// TwinCAT 3 PLC project TcoDataTests
// Title: TcoDataTests
// Company: Vortex.Library
// ProjectVersion: 0.6.0.913
// ProgramVersion: 3.1.4024.12
// libraries:
//   Tc2_Standard, * (Beckhoff Automation GmbH)
//   Tc2_System, * (Beckhoff Automation GmbH)
//   Tc3_Module, * (Beckhoff Automation GmbH)
//   TcoCore, 0.6.0.913 (Vortex.Library)
//   TcoData, 0.6.0.913 (Vortex.Library)
// project tree:
//   DUTs/ SampleDataStructureLevel2.TcDUT, SampleDataStructure.TcDUT
//   / PlcTask.TcTTO
//   POUs/Data/ DataManager.TcPOU, eDataTests.TcDUT, TcoDataExchangeTests.TcPOU
//   POUs/Data/_dummyData/ enumStations.TcDUT, fbAnalogueValueData.TcDUT, stAnalogueProcessData.TcDUT, stCu_Header.TcDUT, stCu_ProcessData.TcDUT, stCu_ProcessDataBase.TcDUT, stEntityHeader.TcDUT, stProcessData.TcDUT
//   POUs/Examples/ eExamplesStates.TcDUT, SandboxData_Plc1.TcDUT, stProcessData_Plc1.TcDUT, stProcessData_Plc2.TcDUT, TcoDataManagerPlc1.TcPOU, TcoDataManagerPlc2.TcPOU, SandboxData.TcDUT, SandboxContext.TcPOU, TcoDataManager.TcPOU
//   POUs/ MAIN.TcPOU, TestDataContext.TcPOU
// (motion and I/O tree: see PLC project tcodata)
// real-time tasks:
//   TASK PlcTask: cycle T#10ms, priority 20, ADS port 350

CONFIGURATION TcoDataTests
    RESOURCE PLC ON TwinCAT3
        TASK PlcTask(INTERVAL := T#10ms, PRIORITY := 20);
        PROGRAM MAIN WITH PlcTask : MAIN;
    END_RESOURCE
END_CONFIGURATION

// ---- DUTs/SampleDataStructureLevel2.TcDUT
TYPE SampleDataStructureLevel2 :
STRUCT
    SampleString : STRING;
    SampleString2 : STRING := '32432423tewtew*-+/';
    SampleInt : INT;
    SampleBool : BOOL;
    SampleBool2 : BOOL := TRUE;
    SampleWString : WSTRING;
    SampleLREAL : LREAL;
END_STRUCT
END_TYPE

// ---- DUTs/SampleDataStructure.TcDUT
TYPE SampleDataStructure :
STRUCT
    SampleString : STRING;
    SampleString2 : STRING := '3retewtertert2342345*-+/';
    SampleInt : INT;
    SampleInt2 : INT := 432;
    SampleBool : BOOL;
    SampleBool2 : BOOL := TRUE;
    SampleWString : WSTRING;
    SampleLREAL : LREAL;
    SampleNestedStructure : SampleDataStructureLevel2;
END_STRUCT
END_TYPE

// ---- POUs/Data/eDataTests.TcDUT
{attribute 'qualified_only'}
{attribute 'strict'}
TYPE eDataTests :
(
    RestoreTasks := 10,
    CreateData := 100,
    UpdateData := 200,
    ReadData := 300,
    DeleteData := 400,
    UpdateDataWithoutChange := 500,
    UpdateDataWithInvalidId := 600,
    ReadDataWithInvlaidId := 700,
    DeleteDataWithInvalidId := 800,
    DataExist := 900,
    CreateOrUpdate := 1000
);
END_TYPE

// ---- POUs/Data/_dummyData/enumStations.TcDUT
{attribute 'qualified_only'}
{attribute 'strict'}
TYPE enumStations :
(
    ST_10 := 10,
    ST_20 := 20,
    ST_30 := 30,
    ST_40 := 40,
    ST_50 := 50,
    ST_60 := 60,
    ST_70 := 70,
    ST_80 := 80,
    ST_90 := 90,
    ST_100 := 100,
    ST_110 := 110,
    ST_120 := 120,
    ST_130 := 130,
    ST_140 := 140,
    ST_150 := 150,
    ST_160 := 160,
    ST_170 := 170,
    ST_180 := 180,
    ST_190 := 190,
    ST_200 := 200
);
END_TYPE

// ---- POUs/Data/_dummyData/fbAnalogueValueData.TcDUT
TYPE fbAnalogueValueData :
STRUCT
    ProcessedData : stAnalogueProcessData;
END_STRUCT
END_TYPE

// ---- POUs/Data/_dummyData/stAnalogueProcessData.TcDUT
TYPE stAnalogueProcessData :
STRUCT
    FailureDescription : STRING;
    Minimum : REAL;
    Maximum : REAL;
END_STRUCT
END_TYPE

// ---- POUs/Data/_dummyData/stCu_Header.TcDUT
TYPE stCu_Header :
STRUCT
    {attribute addProperty Name "<#Next on Passed#>"}
    NextOnPassed : enumStations;
    {attribute addProperty Name "<#Next on Failed#>"}
    NextOnFailed : enumStations;
END_STRUCT
END_TYPE

// ---- POUs/Data/_dummyData/stCu_ProcessData.TcDUT
TYPE stCu_ProcessData EXTENDS stCu_ProcessDataBase :
STRUCT
    {attribute addProperty Name "A_Check_1"}
    A_Check_1 : fbAnalogueValueData;
    {attribute addProperty Name "A_Check_2"}
    A_Check_2 : fbAnalogueValueData;
    {attribute addProperty Name "A_Check_3"}
    A_Check_3 : fbAnalogueValueData;
    {attribute addProperty Name "A_Check_4"}
    A_Check_4 : fbAnalogueValueData;
    {attribute addProperty Name "A_Check_5"}
    A_Check_5 : fbAnalogueValueData;
    {attribute clr [RenderIgnore("Display", "ShadowDisplay")]}
    {attribute addProperty Name "A_Check_6"}
    A_Check_6 : fbAnalogueValueData;
    {attribute clr [RenderIgnore("Control", "ShadowControl")]}
    {attribute addProperty Name "A_Check_7"}
    A_Check_7 : fbAnalogueValueData;
END_STRUCT
END_TYPE

// ---- POUs/Data/_dummyData/stCu_ProcessDataBase.TcDUT
TYPE stCu_ProcessDataBase :
STRUCT
    Header : stCu_Header;
END_STRUCT
END_TYPE

// ---- POUs/Data/_dummyData/stEntityHeader.TcDUT
TYPE stEntityHeader :
STRUCT
    {attribute addProperty Name "Last station"}
    LastStation : enumStations;
    {attribute addProperty Name "Next station"}
    NextStation : enumStations;
END_STRUCT
END_TYPE

// ---- POUs/Data/_dummyData/stProcessData.TcDUT
{attribute wpf [Container(Layout.Tabs)]}
TYPE stProcessData EXTENDS TcoData.TcoEntity :
STRUCT
    {attribute wpf [Container(Layout.Stack)]}
    {attribute addProperty Name "Entity header"}
    EntityHeader ,
    stEntityHeader : BOOL;
    _Modified : DT;
    _Created : DT;
    {attribute wpf [Container(Layout.Stack)]}
    {attribute addProperty Name "Result Data"}
    // {attribute addProperty Name "ST 1"}
    Cu_1 : stCu_ProcessData;
(*Cu_2 : stCu_ProcessData;
    Cu_3 : stCu_ProcessData;
    Cu_4 : stCu_ProcessData;
    Cu_5 : stCu_ProcessData;
    Cu_6 : stCu_ProcessData;
    Cu_7 : stCu_ProcessData;
    Cu_8 : stCu_ProcessData;
    Cu_9 : stCu_ProcessData;
    Cu_10 : stCu_ProcessData;
    *)
END_STRUCT
END_TYPE

// ---- POUs/Examples/eExamplesStates.TcDUT
{attribute 'qualified_only'}
{attribute 'strict'}
TYPE eExamplesStates :
(
    Initialize_1 := 1,
    Initialize_2 := 5,
    Create := 10,
    Update := 20,
    CreateOrUpdate := 30,
    Read := 40,
    Delete := 50,
    Exists := 60
);
END_TYPE

// ---- POUs/Examples/SandboxData_Plc1.TcDUT
//<SandboxData>
// DATA STRUCTURE ELIGIBLE FOR USE WITH TcoDataExchange.
TYPE SandboxData_Plc1 EXTENDS TcoData.TcoEntity :
STRUCT
    sampleData : SampleDataStructure;
    someIntegerPlc1 : INT;
    someStringPlc1 : STRING;
END_STRUCT
END_TYPE
//</SandboxData>

// ---- POUs/Examples/stProcessData_Plc1.TcDUT
{attribute wpf [Container(Layout.Tabs)]}
TYPE stProcessData_Plc1 EXTENDS TcoData.TcoEntity :
STRUCT
    {attribute wpf [Container(Layout.Stack)]}
    {attribute addProperty Name "Entity header"}
    EntityHeader,
    stEntityHeader : BOOL;
    _Modified : DT;
    _Created : DT;
    {attribute wpf [Container(Layout.Stack)]}
    {attribute addProperty Name "Cu1"}
    // {attribute addProperty Name "ST 1"}
    Cu_1 : stCu_ProcessData;
(*Cu_2 : stCu_ProcessData;
    Cu_3 : stCu_ProcessData;
    Cu_4 : stCu_ProcessData;
    Cu_5 : stCu_ProcessData;
    Cu_6 : stCu_ProcessData;
    Cu_7 : stCu_ProcessData;
    Cu_8 : stCu_ProcessData;
    Cu_9 : stCu_ProcessData;
    Cu_10 : stCu_ProcessData;
    *)
END_STRUCT
END_TYPE

// ---- POUs/Examples/stProcessData_Plc2.TcDUT
{attribute wpf [Container(Layout.Tabs)]}
TYPE stProcessData_Plc2 EXTENDS TcoData.TcoEntity :
STRUCT
    {attribute wpf [Container(Layout.Stack)]}
    {attribute addProperty Name "Entity header"}
    EntityHeader,
    stEntityHeader : BOOL;
    _Modified : DT;
    _Created : DT;
    {attribute wpf [Container(Layout.Stack)]}
    // {attribute addProperty Name "ST 1"}
    //Cu_1 : stCu_ProcessData;
    {attribute addProperty Name "Cu2"}
    Cu_2 : stCu_ProcessData;
(*Cu_3 : stCu_ProcessData;
    Cu_4 : stCu_ProcessData;
    Cu_5 : stCu_ProcessData;
    Cu_6 : stCu_ProcessData;
    Cu_7 : stCu_ProcessData;
    Cu_8 : stCu_ProcessData;
    Cu_9 : stCu_ProcessData;
    Cu_10 : stCu_ProcessData;
    *)
END_STRUCT
END_TYPE

// ---- POUs/Examples/SandboxData.TcDUT
//<SandboxData>
// DATA STRUCTURE ELIGIBLE FOR USE WITH TcoDataExchange.
TYPE SandboxData EXTENDS TcoData.TcoEntity :
STRUCT
    sampleData : SampleDataStructure;
    someInteger : INT;
    someString : STRING;
END_STRUCT
END_TYPE
//</SandboxData>

// ---- POUs/MAIN.TcPOU
PROGRAM MAIN
VAR
    dataTests : TestDataContext;
    sandbox : SandboxContext;
END_VAR

dataTests.ProbeRun();
sandbox.Run();

END_PROGRAM

// ---- POUs/TestDataContext.TcPOU
FUNCTION_BLOCK TestDataContext EXTENDS TcoCore._internals_TcoContext
VAR
    DataTests : TcoDataExchangeTests(THIS^);
    _identifier : STRING;
    _restoreTasksDone : BOOL;
    _createDataDone : BOOL;
    _updateDataDone : BOOL;
    _readDataDone : BOOL;
    _deleteDataDone : BOOL;
    _updateDataWithoutChangeDone : BOOL;
    _updateDataWithInvalidIdDone : BOOL;
    _readDataWithInvlaidIdDone : BOOL;
    _deleteDataWithInvalidIdDone : BOOL;
    _dataExistsDone : BOOL;
    _createOrUpdateDone : BOOL;
END_VAR

METHOD PROTECTED Main
VAR_INST
    RunCreate : BOOL;
END_VAR
DataTests();

CASE THIS^._testId OF
    eDataTests.RestoreTasks:
        DataTests.DataManager._createTask.Restore();
        DataTests.DataManager._readTask.Restore();
        DataTests.DataManager._updateTask.Restore();
        DataTests.DataManager._deleteTask.Restore();
        DataTests.DataManager._idExistsTask.Restore();
        DataTests.DataManager._createOrUpdateTask.Restore();
    eDataTests.CreateData:
        _createDataDone := DataTests.Create(_identifier);
    eDataTests.UpdateData:
        _updateDataDone := DataTests.Update(_identifier);
    eDataTests.ReadData:
        _readDataDone := DataTests.Read(_identifier);
    eDataTests.DeleteData:
        _deleteDataDone := DataTests.Delete(_identifier);
    eDataTests.UpdateDataWithoutChange:
        _updateDataWithoutChangeDone := DataTests.UpdateDataWithoutChange(_identifier);
    eDataTests.UpdateDataWithInvalidId:
        _updateDataWithInvalidIdDone := DataTests.UpdateDataWithInvalidId();
    eDataTests.ReadDataWithInvlaidId:
        _readDataWithInvlaidIdDone := DataTests.ReadDataWithInvlaidId();
    eDataTests.DeleteDataWithInvalidId:
        _deleteDataWithInvalidIdDone := DataTests.DeleteDataWithInvalidId();
    eDataTests.DataExist:
        _dataExistsDone := DataTests.ExistsTest(_identifier);
    eDataTests.CreateOrUpdate:
        _createOrUpdateDone := DataTests.CreateOrUpdate(_identifier);
END_CASE
END_METHOD

END_FUNCTION_BLOCK

// ---- POUs/Data/TcoDataExchangeTests.TcPOU
FUNCTION_BLOCK TcoDataExchangeTests EXTENDS TcoCore.TcoObject
VAR
    DataManager : DataManager(THIS^);
END_VAR

DataManager();

{attribute 'TcRpcEnable'}
METHOD Create : BOOL
VAR_INPUT
    Identifier : STRING;
END_VAR
DataManager.Data.Cu_1.A_Check_1.ProcessedData.FailureDescription := 'Writing failure from PLC';
DataManager.Data.Cu_1.A_Check_1.ProcessedData.Maximum := 10;
DataManager.Data.Cu_1.A_Check_1.ProcessedData.Minimum := 5;
Create := DataManager.Create(Identifier).Done;
END_METHOD

METHOD CreateOrUpdate : BOOL
VAR_INPUT
    Identifier : STRING;
END_VAR
CreateOrUpdate := DataManager.CreateOrUpdate(Identifier).Done;
END_METHOD

METHOD Delete : BOOL
VAR_INPUT
    Identifier : STRING;
END_VAR
Delete := DataManager.Delete(Identifier).Done;
END_METHOD

METHOD DeleteDataWithInvalidId : BOOL
VAR_INPUT
END_VAR
DeleteDataWithInvalidId := DataManager.Delete(ULINT_TO_STRING(Context.RealTimeClock.TickClock())).Done;
END_METHOD

METHOD ExistsTest : BOOL
VAR_INPUT
    inIdentifier : STRING(255);
END_VAR
ExistsTest := THIS^.DataManager.Exists(inIdentifier).Done;
END_METHOD

METHOD Read : BOOL
VAR_INPUT
    Identifier : STRING;
END_VAR
Read := DataManager.Read(Identifier).Done;
END_METHOD

METHOD ReadDataWithInvlaidId : BOOL
VAR_INPUT
END_VAR
ReadDataWithInvlaidId := DataManager.Read(ULINT_TO_STRING(Context.RealTimeClock.TickClock())).Error;
END_METHOD

METHOD Update : BOOL
VAR_INPUT
    Identifier : STRING;
END_VAR
DataManager.Data.Cu_1.A_Check_1.ProcessedData.FailureDescription := 'Updated failure from PLC';
DataManager.Data.Cu_1.A_Check_1.ProcessedData.Maximum := 20;
DataManager.Data.Cu_1.A_Check_1.ProcessedData.Minimum := 10;
Update := DataManager.Update(Identifier).Done;
END_METHOD

METHOD UpdateDataWithInvalidId : BOOL
VAR_INPUT
END_VAR
UpdateDataWithInvalidId := DataManager.Update(ULINT_TO_STRING(Context.RealTimeClock.TickClock())).Error;
END_METHOD

METHOD UpdateDataWithoutChange : BOOL
VAR_INPUT
    Identifier : STRING;
END_VAR
UpdateDataWithoutChange := DataManager.Create(Identifier).Done AND_THEN DataManager.Update(Identifier).Done;
END_METHOD

END_FUNCTION_BLOCK

// ---- POUs/Data/DataManager.TcPOU
FUNCTION_BLOCK DataManager EXTENDS TcoData.TcoDataExchange
VAR
    _data : stProcessData;
END_VAR

SUPER^();

PROPERTY Data : REFERENCE TO stProcessData
GET
DATA REF= _data;
END_GET
END_PROPERTY

END_FUNCTION_BLOCK

// ---- POUs/Examples/SandboxContext.TcPOU
//<Declaration>
FUNCTION_BLOCK SandboxContext EXTENDS TcoCore.TcoContext
VAR
    DataManager : TcoDataManager(THIS^);
    DataManagerFragmented : TcoDataManager(THIS^);
    DataManagerPlc1 : TcoDataManagerPlc1(THIS^);
    DataManagerPlc2 : TcoDataManagerPlc2(THIS^);
    //	DataManagerFragmentedPlc1 : TcoDataManagerPlc1(THIS^);
END_VAR
//</Declaration>
VAR
    _state : eExamplesStates;
    recordId_1 : STRING;
    recordId_2 : STRING;
    _invokeSearch : BOOL;
    _filteringById : STRING;
END_VAR

(*~
    <docu>
        <summary>
            Main method of the TcoContext. This is the entry point of any control logic that belongs to this context.
            The call of this method is ensured by calling the <c>InstanceName.Run()</c> method, and it must not be called explicitly.
            This method is abstract, and it must be overridden in derived block.
        </summary>
    </docu>
~*)
METHOD PROTECTED Main
// Context logging configuration
Context.Environment.Messaging.MessageDigestMethod := eMessageDigestMethod.CRC32;
Context.Environment.Messaging.MessengerLoggingMethod := eMessengerLogMethod.OnEventRisen;
//<CyclicalDataMangerCall>
// Cyclical data manage call.
DataManager();
DataManagerFragmented();
DataManagerPlc1();
DataManagerPlc2();
//</CyclicalDataMangerCall>
recordId_1 := 'scoundrel';
recordId_2 := 'knight';

CASE _state OF
    eExamplesStates.Initialize_1:
        IF (DataManager.Exists(recordId_1).Done) THEN
            IF (DataManager.Exists(recordId_1).Exists) THEN
                IF (DataManager.Delete(recordId_1).Done) THEN
                    DataManager.Messenger.Build().Append('Record ').Append(recordId_1).Append(' deleted.').As().AsInfo();
                END_IF;
            END_IF
        END_IF
    eExamplesStates.Initialize_2:
        IF (DataManager.Exists(recordId_2).Done) THEN
            IF (DataManager.Exists(recordId_2).Exists) THEN
                IF (DataManager.Delete(recordId_2).Done) THEN
                    DataManager.Messenger.Build().Append('Record ').Append(recordId_2).Append(' deleted.').As().AsInfo();
                END_IF;
            END_IF
        END_IF
    eExamplesStates.Create:
        //<CreateCodeExample>
        // Will create new entry into repository with data contained in the `_data`
        IF (DataManager.Create(recordId_1).Done) THEN
            DataManager.Messenger.Build().Append('Record ').Append(recordId_1).Append(' created.').As().AsInfo();
        END_IF;
    //</CreateCodeExample>
    eExamplesStates.Update:
        // <UpdateCodeExample>
        DataManager.Data.sampleData.SampleInt := 33;
        DataManager.Data.sampleData.SampleString := 'Max';
        DataManager.Data.sampleData.SampleNestedStructure.SampleLREAL := 1;

        IF (DataManager.Update(recordId_1).Done) THEN
            DataManager.Messenger.Build().Append('Record ').Append(recordId_1).Append(' updated.').As().AsInfo();
        END_IF;
    // </UpdateCodeExample>
    eExamplesStates.CreateOrUpdate:
        // <CreateOrUpdateCodeExample>
        DataManager.Data.sampleData.SampleInt := 44;
        DataManager.Data.sampleData.SampleString := 'Lewis';
        DataManager.Data.sampleData.SampleNestedStructure.SampleLREAL := 7;

        IF (DataManager.CreateOrUpdate(recordId_2).Done) THEN
            DataManager.Messenger.Build().Append('Record ').Append(recordId_2).Append(' updated/created.').As().AsInfo();
        END_IF;
    // <CreateOrUpdateCodeExample>
    eExamplesStates.Read:
        // <ReadCodeExample>
        IF (DataManager.Read(recordId_1).Done) THEN
            DataManager.Messenger.Build()
                .Append('Record ')
                .Append(recordId_1)
                .Append(' read.')
                .AppendAny(DataManager.Data.sampleData.SampleInt)
                .Append(';')
                .Append(DataManager.Data.sampleData.SampleString)
                .Append(';')
                .AppendAny(DataManager.Data.sampleData.SampleNestedStructure.SampleLREAL)
                .As().AsInfo();
        END_IF;
    // </ReadCodeExample>
    eExamplesStates.Delete:
        // <DeleteCodeExample>
        IF (DataManager.Delete(recordId_1).Done) THEN
            DataManager.Messenger.Build().Append('Record ').Append(recordId_1).Append(' deleted.').As().AsInfo();
        END_IF;
    // </DeleteCodeExample>
    eExamplesStates.Exists:
        // <ExistsCodeExample>
        IF (DataManager.Exists(recordId_2).Done) THEN
            DataManager.Messenger.Clear();

            IF (DataManager.Exists(recordId_2).Exists) THEN
                DataManager.Messenger.Build().Append('Record ').Append(recordId_2).Append(' exists.').As().AsInfo();
            ELSE
                DataManager.Messenger.Build().Append('Record ').Append(recordId_2).Append(' does not exists.').As().AsInfo();
            END_IF
        END_IF
    // </ExistsCodeExample>
END_CASE
END_METHOD

END_FUNCTION_BLOCK

// ---- POUs/Examples/TcoDataManager.TcPOU
//<DataManagerDeclarations>
// Function block for data maipulation must extend from TcoData.TcoDataExchange.
FUNCTION_BLOCK TcoDataManager EXTENDS TcoData.TcoDataExchange
VAR
    // This is the structure that contains the actual data we will work with. The `STRUCT` must extend `TcoData.TcoEntity`
    _data : SandboxData;
END_VAR
//</DataManagerDeclarations>

//----------------------------------
//<DataManagerSuperCall>
// IMPLEMENTATION BODY OF FUNCTION BLOCK
// IMPORTANT: SUPER CALL HERE IS REQUIRED TO CALL THE DATA MANAGER TASKS!!!
SUPER^();
//</DataManagerSuperCall>
//----------------------------------

PROPERTY Data : REFERENCE TO SandboxData
GET
Data REF= _data;
END_GET
END_PROPERTY

END_FUNCTION_BLOCK

// ---- POUs/Examples/TcoDataManagerPlc1.TcPOU
//<DataManagerDeclarations>
// Function block for data maipulation must extend from TcoData.TcoDataExchange.
FUNCTION_BLOCK TcoDataManagerPlc1 EXTENDS TcoData.TcoDataExchange
VAR
    // This is the structure that contains the actual data we will work with. The `STRUCT` must extend `TcoData.TcoEntity`
    _data : stProcessData_Plc1;
END_VAR
//</DataManagerDeclarations>

//----------------------------------
//<DataManagerSuperCall>
// IMPLEMENTATION BODY OF FUNCTION BLOCK
// IMPORTANT: SUPER CALL HERE IS REQUIRED TO CALL THE DATA MANAGER TASKS!!!
SUPER^();
//</DataManagerSuperCall>
//----------------------------------

PROPERTY Data : REFERENCE TO stProcessData_Plc1
GET
Data REF= _data;
END_GET
END_PROPERTY

END_FUNCTION_BLOCK

// ---- POUs/Examples/TcoDataManagerPlc2.TcPOU
//<DataManagerDeclarations>
// Function block for data maipulation must extend from TcoData.TcoDataExchange.
FUNCTION_BLOCK TcoDataManagerPlc2 EXTENDS TcoData.TcoDataExchange
VAR
    // This is the structure that contains the actual data we will work with. The `STRUCT` must extend `TcoData.TcoEntity`
    _data : stProcessData_Plc2;
END_VAR
//</DataManagerDeclarations>

//----------------------------------
//<DataManagerSuperCall>
// IMPLEMENTATION BODY OF FUNCTION BLOCK
// IMPORTANT: SUPER CALL HERE IS REQUIRED TO CALL THE DATA MANAGER TASKS!!!
SUPER^();
//</DataManagerSuperCall>
//----------------------------------

PROPERTY Data : REFERENCE TO stProcessData_Plc2
GET
Data REF= _data;
END_GET
END_PROPERTY

END_FUNCTION_BLOCK
